(*
SPDX-FileCopyrightText: Â© 2026 Oleksandr Tiutyk <trofimich@gmail.com>
SPDX-License-Identifier: MIT
License: https://opensource.org/license/mit
*)

(*!
<summary>Represents an automation component capable of operating in simulation mode.</summary>
<description>
Provides read access to the active simulation mode status.
</description>
*)

INTERFACE ISimulatable EXTENDS TOF_Core.IObject

(*!
<summary>Gets whether simulation mode is currently active.</summary>
*)
{attribute 'monitoring' := 'call'}
PROPERTY SimulationMode : BOOL
GET
END_GET
END_PROPERTY

END_INTERFACE

(* stored: Version 1.1.0.1
   Itf ISimulatable: Id {64def839-9c7f-49fb-bb6c-6e139237e3fc}
   Property SimulationMode: Id {f5dfb847-33cc-4380-a1cf-0d2edbb1a6ef}
   Get Get: Id {26bbacea-8cbd-4c03-a1df-2721a1043836} *)
